Staubli VAL3: getView.pgx

public program getView(bool& x_bView[])
begin
  if nBottomX==38
    x_bView=true
  else
    x_bView=false
  endIf
end
